{attribute 'linkalways'} 
{attribute 'no_explicit_call' := 'This FB is a CLASS and must be accessed using methods or properties'}
{attribute 'enable_dynamic_creation'}
FUNCTION_BLOCK _HRESULT EXTENDS AliasDatatypeBase
VAR
	localData : HRESULT;
	activeData : REFERENCE TO HRESULT REF= localData;
	aliasBaseType : _DINT(localData);
END_VAR

PROPERTY PUBLIC Address : PVOID
GET
Address := ADR(activeData);
END_GET
END_PROPERTY

METHOD PUBLIC ClearReference
VAR_INPUT
END_VAR
activeData REF= localData;
SetBaseTypeReference();
END_METHOD

METHOD PUBLIC Clone : I_Datatype
VAR
    pClone : POINTER TO _HRESULT;
END_VAR
pClone := __NEW(_HRESULT(InitialValue := Value));
Clone := pClone^;
END_METHOD

METHOD FB_init : BOOL
VAR_INPUT
	bInitRetains : BOOL; // if TRUE, the retain variables are initialized (warm start / cold start)
	bInCopyCode : BOOL;  // if TRUE, the instance afterwards gets moved into the copy code (online change)
	InitialValue : HRESULT;
END_VAR
localData := InitialValue;
SetBaseTypeReference();
AddBaseType(aliasBaseType);
END_METHOD

PROPERTY PUBLIC Identifier : T_MAXSTRING
GET
Identifier := 'HRESULT';
END_GET
END_PROPERTY

METHOD PUBLIC MakeReferenceTo
VAR_INPUT
	ReferenceTarget : REFERENCE TO HRESULT;
END_VAR
activeData REF= ReferenceTarget;
SetBaseTypeReference();
END_METHOD

METHOD PROTECTED SetBaseTypeReference
VAR_INPUT
END_VAR
aliasBaseType.MakeReferenceTo(activeData);
END_METHOD

PROPERTY PUBLIC Size : UDINT
GET
Size := SIZEOF(activeData);
END_GET
END_PROPERTY

METHOD TryMakeReferenceTo : BOOL
VAR_INPUT
	Target : I_Datatype;
END_VAR
VAR
	targetAsAlias : I_AliasDatatype;
	pTargetData : POINTER TO HRESULT;
END_VAR
IF NOT Target.TryResolveAsAliasType(targetAsAlias) THEN
	RETURN;
END_IF

IF targetAsAlias.Identifier <> Identifier THEN
	RETURN;
END_IF

pTargetData := Target.Address;
activeData REF= pTargetData^;
SetBaseTypeReference();
TryMakeReferenceTo := TRUE;
END_METHOD

PROPERTY PUBLIC Value : HRESULT
GET
Value := activeData;
END_GET
SET
activeData := Value;
END_SET
END_PROPERTY

END_FUNCTION_BLOCK

(* stored: Version 1.1.0.1, ProductVersion 3.1.4024.12
   POU _HRESULT: Id {812bad4a-7bd2-0ca8-1e32-53ad4f652147}, SpecialFunc None
   Folder Constructor: Id {c86d702f-77a8-0c2d-2692-85b706f92094}
   Folder Protected: Id {e16fea1f-f592-091f-2024-44bbaa215477}
   Property Address: Id {eaea8ce2-d780-069a-2354-b9040dbfdf59}
   Get Get: Id {9ca66335-2df6-0b97-035a-cfdc96d663e4}
   Method ClearReference: Id {3b3306cf-50f2-0e29-0162-910cb3f73574}
   Method Clone: Id {3e05ef98-5afd-4b49-b284-8e3d2d8200da}
   Method FB_init: Id {86e1a4c2-65f3-05c8-1412-88763e434d4e}
   Property Identifier: Id {783e0e3e-7447-0c8f-3ba4-419752f4a16d}
   Get Get: Id {48ca57da-3d4d-0ccb-0db1-4ab3be926971}
   Method MakeReferenceTo: Id {b812282b-13cf-0ccc-1aff-702feb80c71d}
   Method SetBaseTypeReference: Id {68a695f5-ff13-0dcc-1466-991b2c518bab}
   Property Size: Id {78fc7983-bbf0-072e-3bed-9c1f413ab6ff}
   Get Get: Id {1ef01c66-9a0c-0188-28d6-15ce2d32f45d}
   Method TryMakeReferenceTo: Id {43bcd589-1009-0f1a-3a87-0d5bc8645b2a}
   Property Value: Id {85c486dd-d750-0c76-00cb-4c376724f1d2}
   Get Get: Id {d04c4bc3-8e0b-04d3-3b2c-700ab80225ae}
   Set Set: Id {44e9d433-2f91-0b46-3692-b60205dde3fd} *)
